Staubli VAL3: PROG.dtx

public progItem pProg{}
  [0001]
    InstrItem iEvent[5]
      [0]
        string sData = "qujian"
        string sType = "TRAJ"
      [1]
        string sData = "langyong"
        string sType = "TRAJ"
      [2]
        string sData = "cuigan1"
        string sType = "JPOINT"
      [3]
        string sData = "cuigan2"
        string sType = "TRAJ"
      [4]
        string sData = "home"
        string sType = "HOME"
    string sID = "0001"
  [001 prd1]
    InstrItem iEvent[8]
      [0]
        string sData = "qujian"
        string sType = "TRAJ"
      [1]
        string sData = "langyong"
        string sType = "TRAJ"
      [2]
        string sData = "cuigan1"
        string sType = "JPOINT"
      [3]
        string sData = "cuigan1"
        string sType = "TRAJ"
      [4]
        string sData = "cuigan2"
        string sType = "JPOINT"
      [5]
        string sData = "cuigan2"
        string sType = "TRAJ"
      [6]
        string sData = "huilu"
        string sType = "JPOINT"
      [7]
        string sData = "home"
        string sType = "HOME"
    string sID = "001 prd1"
  [002 prd2]
    InstrItem iEvent
      [0]
        string sData = "qujian"
        string sType = "TRAJ"
    string sID = "002 prd2"
  [HOME1]
    InstrItem iEvent
      [0]
        string sData
        string sType
    string sID = "HOME1"
  [HOME2]
    InstrItem iEvent
      [0]
        string sData
        string sType
    string sID = "HOME2"
